FUNCTION_BLOCK HMI_BUTTONS_VV (* Human machine interface for input *)
  (* Standard: 61499-2 *)
  (* Version 0.1, 2002-01-08, JHC, Rockwell Automation, Added DLY FB as example. *)
  (* Version 0.0, 2000-05-27, JHC, Rockwell Automation *)
  (* Compiler header: package fb.rt.festo1;import fb.rt.swing.*;import fb.rt.hmi.*; *)
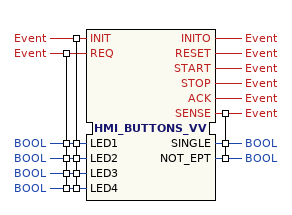
  EVENT_INPUT
    INIT WITH LED1, LED2, LED3, LED4; (* Initialization Request *)
    REQ WITH LED1, LED2, LED3, LED4;
  END_EVENT
  EVENT_OUTPUT
    INITO; (* Initialization Confirm *)
    RESET; (* Execution Confirmation *)
    START; (* Execution Confirmation *)
    STOP; (* Execution Confirmation *)
    ACK; (* Execution Confirmation *)
    SENSE WITH SINGLE, NOT_EPT; (* Execution Confirmation *)
  END_EVENT
  VAR_INPUT
    LED1 : BOOL;
    LED2 : BOOL;
    LED3 : BOOL;
    LED4 : BOOL;
  END_VAR
  VAR_OUTPUT
    SINGLE : BOOL; (* Output event qualifier *)
    NOT_EPT : BOOL; (* Output event qualifier *)
  END_VAR
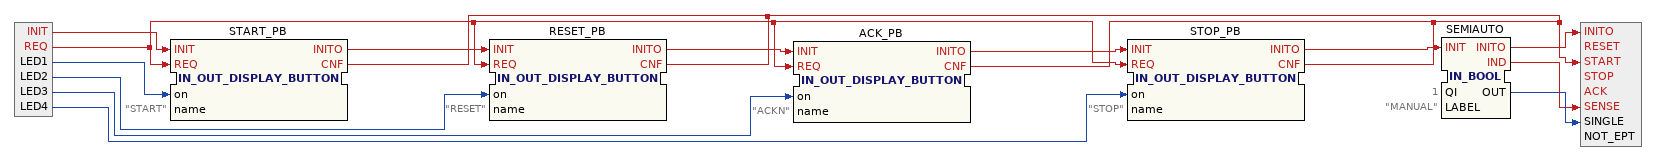
  FBS
    START_PB : IN_OUT_DISPLAY_BUTTON(name := "START");
    RESET_PB : IN_OUT_DISPLAY_BUTTON(name := "RESET");
    STOP_PB : IN_OUT_DISPLAY_BUTTON(name := "STOP");
    ACK_PB : IN_OUT_DISPLAY_BUTTON(name := "ACKN");
    SEMIAUTO : IN_BOOL(QI := 1, LABEL := "MANUAL");
  END_FBS
  EVENT_CONNECTIONS
    INIT TO START_PB.INIT;
    START_PB.INITO TO RESET_PB.INIT;
    RESET_PB.INITO TO ACK_PB.INIT;
    ACK_PB.INITO TO STOP_PB.INIT;
    STOP_PB.INITO TO SEMIAUTO.INIT;
    SEMIAUTO.INITO TO INITO;
    SEMIAUTO.IND TO SENSE;
    REQ TO START_PB.REQ;
    REQ TO RESET_PB.REQ;
    REQ TO ACK_PB.REQ;
    REQ TO STOP_PB.REQ;
    START_PB.CNF TO START;
    RESET_PB.CNF TO START;
    ACK_PB.CNF TO START;
    STOP_PB.CNF TO START;
  END_CONNECTIONS
  DATA_CONNECTIONS
    SEMIAUTO.OUT TO SINGLE;
    LED1 TO START_PB.on;
    LED2 TO RESET_PB.on;
    LED3 TO ACK_PB.on;
    LED4 TO STOP_PB.on;
  END_CONNECTIONS
END_FUNCTION_BLOCK
